PROGRAM Interlocks_to_Main_Line
VAR
	RibMachineReady: BOOL;
	
	
	
END_VAR

// NETWORK 1

END_PROGRAM

(* stored: Version 1.1.0.1, ProductVersion 3.1.4024.12
   POU Interlocks_to_Main_Line: Id {fc071314-457f-455f-a9b7-0b493a5df2e8}, SpecialFunc None *)
